FUNCTION_BLOCK minMax (* Basic Function Block Type *)
  (* Standard: 61499-2 *)
  (* Version 0.0, 11.10.2011, herrric, nxtControl GmbH, Template *)
  PACKAGE Loytec.HVAC;
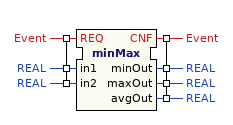
  EVENT_INPUT
    REQ WITH in1, in2; (* Normal Execution Request *)
  END_EVENT
  EVENT_OUTPUT
    CNF WITH minOut, maxOut, avgOut; (* Execution Confirmation *)
  END_EVENT
  VAR_INPUT
    in1 : REAL; (* Input event qualifier *)
    in2 : REAL;
  END_VAR
  VAR_OUTPUT
    minOut : REAL; (* Output event qualifier *)
    maxOut : REAL;
    avgOut : REAL;
  END_VAR
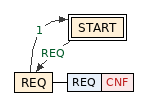
  EC_STATES
    START; (* Initial State *)
    REQ : REQ -> CNF; (* Normal execution *)
  END_STATES
  EC_TRANSITIONS
    START TO REQ := REQ;
    REQ TO START := 1;
  END_TRANSITIONS
  ALGORITHM REQ IN ST: (* Normally executed algorithm *)
minOut := MIN(in1, in2);
maxOut := MAX(in1, in2);
avgOut := (in1 + in2) / 2;
  END_ALGORITHM
END_FUNCTION_BLOCK
